(* Logix 5000 project; controller SX_V040001_C001 vendor 1 type 14 code 77 rev 16.23; software revision 16.04; part 11 of 35 *)
(* tags used below, declared in another part *)
   ALL_KINDS : INT[90];
   Basic : INT;
   DRIVE : INT[32];
   DRIVE_INTERVAL : INT[8];
   EMPTYING : INT[18];
   G_AOutput : DINT[8];
   G_DInput : DINT[3];
   G_DOutput : DINT[3];
   METERING : INT[44];
   METERING_PULSE : DINT[14];
   negi_param398 : DINT;
   NOTDOS : INT[6];
   PARAMETER : INT[501];
   T_ACT_DATA_RESET : TIMER;
   T_CHOCO_PRESS_LOW : TIMER;
   T_DEL_DATA : TIMER;
   T_OUTLET_CLOSE : TIMER;
   T_RUN_OUT_CHOCOPUMP : TIMER;
(* MainProgram, continued *)

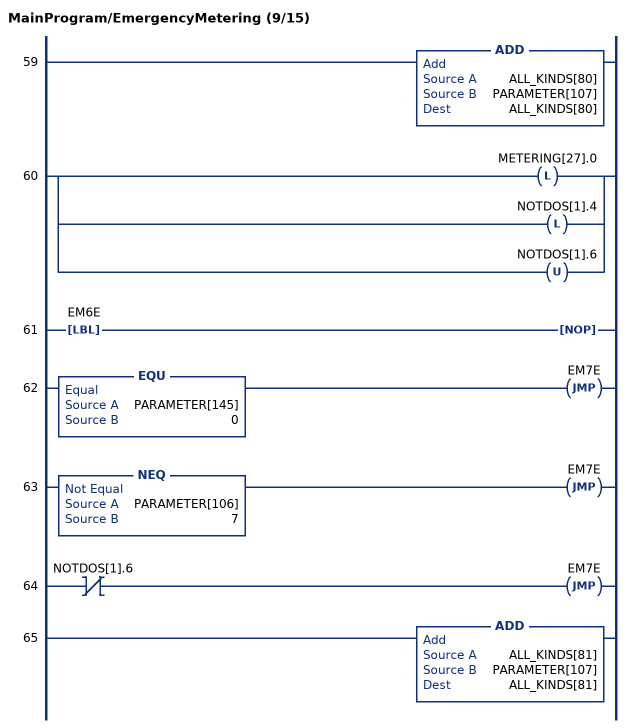
   [picture p232: MainProgram/EmergencyMetering rungs 59-65]
   59: ADD(ALL_KINDS[80],PARAMETER[107],ALL_KINDS[80]);
   60: [OTL(METERING[27].0) ,OTL(NOTDOS[1].4) ,OTU(NOTDOS[1].6) ];
   61: LBL(EM6E)NOP();
   62: EQU(PARAMETER[145],0)JMP(EM7E);
   63: NEQ(PARAMETER[106],7)JMP(EM7E);
   64: XIO(NOTDOS[1].6)JMP(EM7E);
   65: ADD(ALL_KINDS[81],PARAMETER[107],ALL_KINDS[81]);
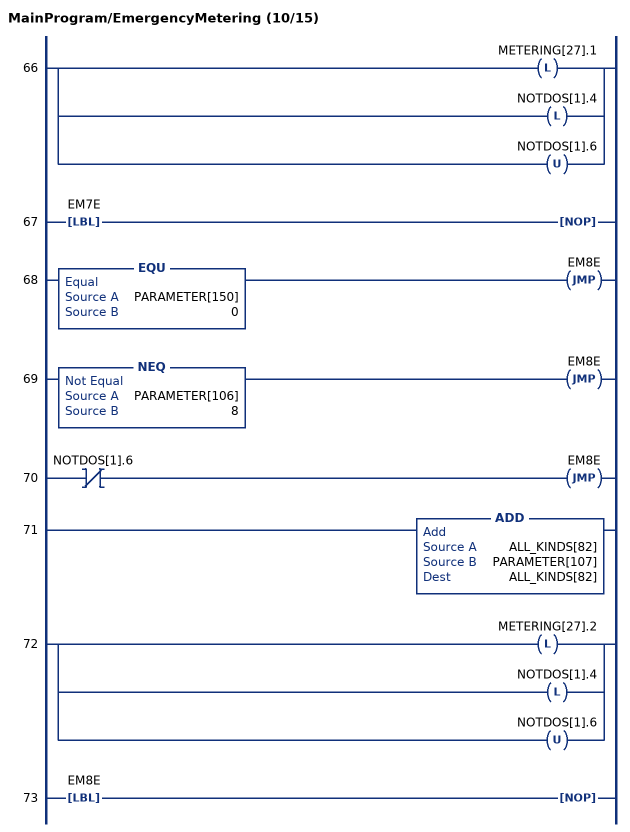
   66: [OTL(METERING[27].1) ,OTL(NOTDOS[1].4) ,OTU(NOTDOS[1].6) ];
   67: LBL(EM7E)NOP();
   68: EQU(PARAMETER[150],0)JMP(EM8E);
   69: NEQ(PARAMETER[106],8)JMP(EM8E);
   70: XIO(NOTDOS[1].6)JMP(EM8E);
   71: ADD(ALL_KINDS[82],PARAMETER[107],ALL_KINDS[82]);
   72: [OTL(METERING[27].2) ,OTL(NOTDOS[1].4) ,OTU(NOTDOS[1].6) ];
   73: LBL(EM8E)NOP();
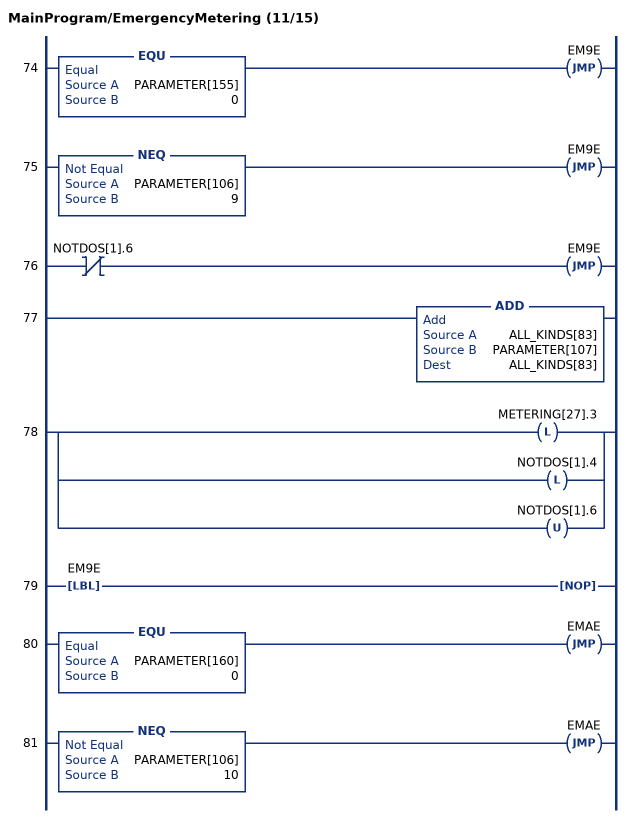
   74: EQU(PARAMETER[155],0)JMP(EM9E);
   75: NEQ(PARAMETER[106],9)JMP(EM9E);
   76: XIO(NOTDOS[1].6)JMP(EM9E);
   77: ADD(ALL_KINDS[83],PARAMETER[107],ALL_KINDS[83]);
   78: [OTL(METERING[27].3) ,OTL(NOTDOS[1].4) ,OTU(NOTDOS[1].6) ];
   79: LBL(EM9E)NOP();
   80: EQU(PARAMETER[160],0)JMP(EMAE);
   81: NEQ(PARAMETER[106],10)JMP(EMAE);
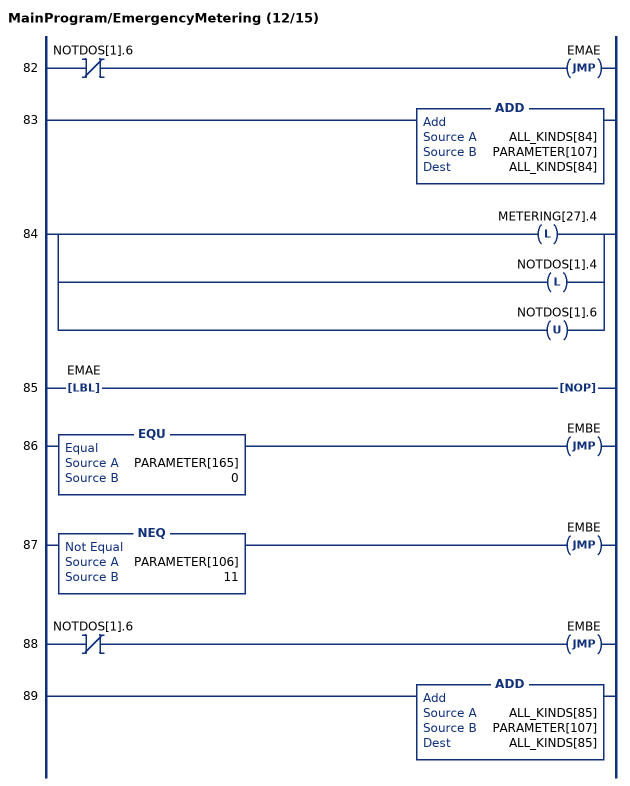
   82: XIO(NOTDOS[1].6)JMP(EMAE);
   83: ADD(ALL_KINDS[84],PARAMETER[107],ALL_KINDS[84]);
   84: [OTL(METERING[27].4) ,OTL(NOTDOS[1].4) ,OTU(NOTDOS[1].6) ];
   85: LBL(EMAE)NOP();
   86: EQU(PARAMETER[165],0)JMP(EMBE);
   87: NEQ(PARAMETER[106],11)JMP(EMBE);
   88: XIO(NOTDOS[1].6)JMP(EMBE);
   89: ADD(ALL_KINDS[85],PARAMETER[107],ALL_KINDS[85]);
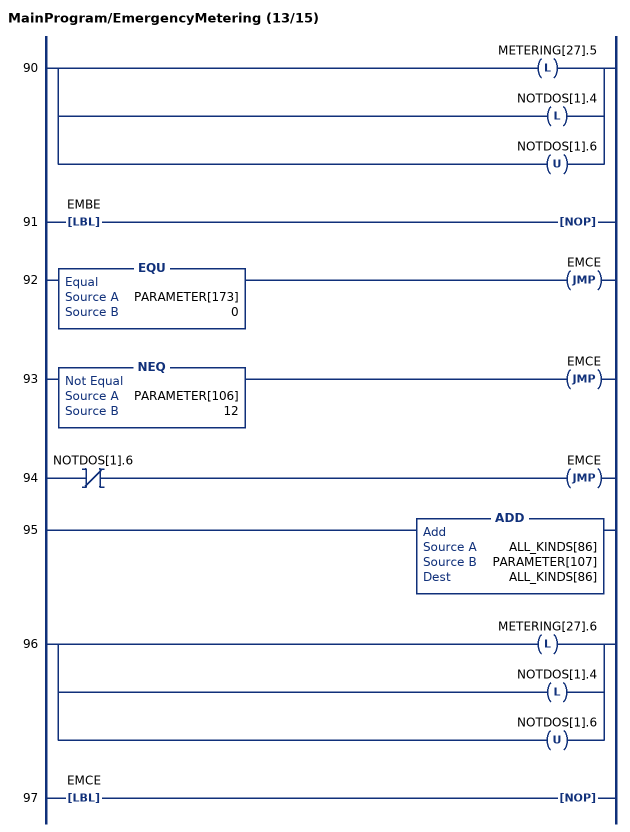
   90: [OTL(METERING[27].5) ,OTL(NOTDOS[1].4) ,OTU(NOTDOS[1].6) ];
   91: LBL(EMBE)NOP();
   92: EQU(PARAMETER[173],0)JMP(EMCE);
   93: NEQ(PARAMETER[106],12)JMP(EMCE);
   94: XIO(NOTDOS[1].6)JMP(EMCE);
   95: ADD(ALL_KINDS[86],PARAMETER[107],ALL_KINDS[86]);
   96: [OTL(METERING[27].6) ,OTL(NOTDOS[1].4) ,OTU(NOTDOS[1].6) ];
   97: LBL(EMCE)NOP();
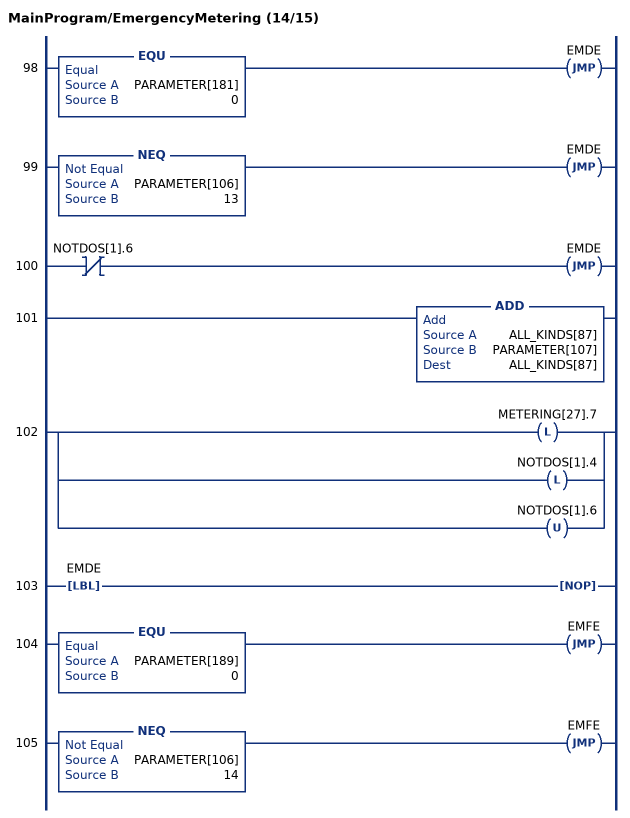
   98: EQU(PARAMETER[181],0)JMP(EMDE);
   99: NEQ(PARAMETER[106],13)JMP(EMDE);
   100: XIO(NOTDOS[1].6)JMP(EMDE);
   101: ADD(ALL_KINDS[87],PARAMETER[107],ALL_KINDS[87]);
   102: [OTL(METERING[27].7) ,OTL(NOTDOS[1].4) ,OTU(NOTDOS[1].6) ];
   103: LBL(EMDE)NOP();
   104: EQU(PARAMETER[189],0)JMP(EMFE);
   105: NEQ(PARAMETER[106],14)JMP(EMFE);
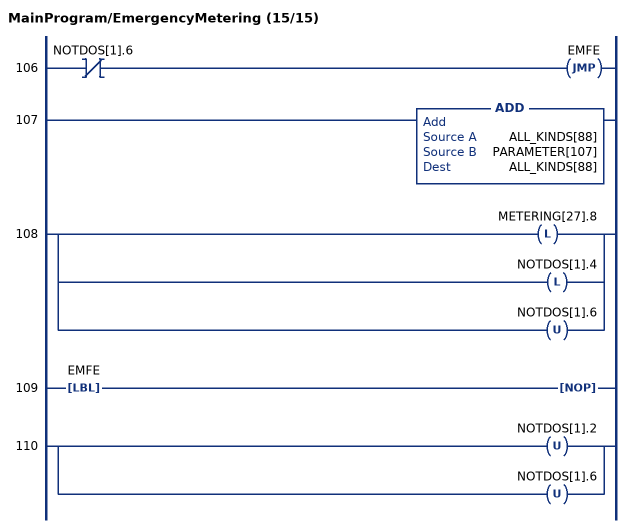
   106: XIO(NOTDOS[1].6)JMP(EMFE);
   107: ADD(ALL_KINDS[88],PARAMETER[107],ALL_KINDS[88]);
   108: [OTL(METERING[27].8) ,OTL(NOTDOS[1].4) ,OTU(NOTDOS[1].6) ];
   109: LBL(EMFE)NOP();
   110: [OTU(NOTDOS[1].2) ,OTU(NOTDOS[1].6) ];
END_ROUTINE

ROUTINE Emptying   (* ladder *)
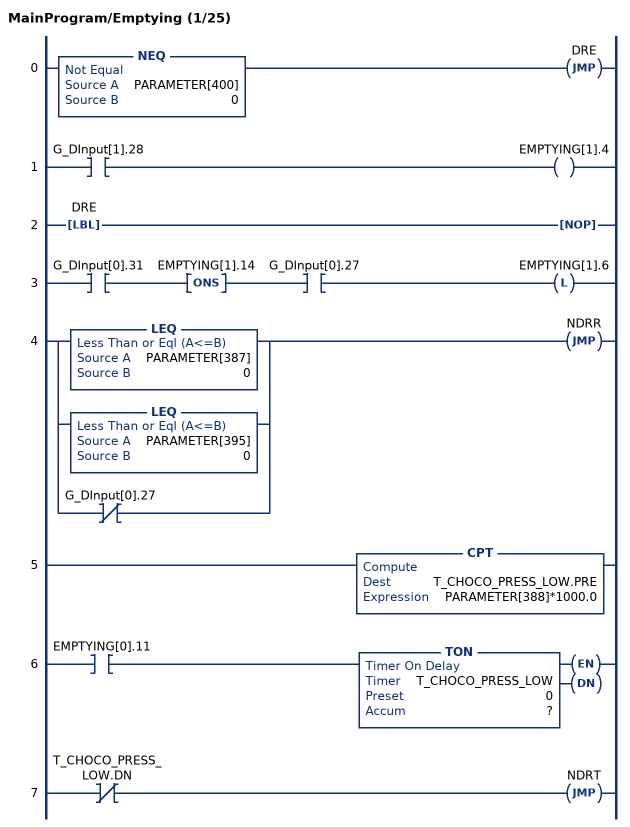
   0: NEQ(PARAMETER[400],0)JMP(DRE);
   1: XIC(G_DInput[1].28)OTE(EMPTYING[1].4);
   2: LBL(DRE)NOP();
   3: XIC(G_DInput[0].31)ONS(EMPTYING[1].14)XIC(G_DInput[0].27)OTL(EMPTYING[1].6);
   4: [LEQ(PARAMETER[387],0) ,LEQ(PARAMETER[395],0) ,XIO(G_DInput[0].27) ]JMP(NDRR);
   5: CPT(T_CHOCO_PRESS_LOW.PRE,PARAMETER[388]*1000.0);
   6: XIC(EMPTYING[0].11)TON(T_CHOCO_PRESS_LOW,?,?);
   7: XIO(T_CHOCO_PRESS_LOW.DN)JMP(NDRT);
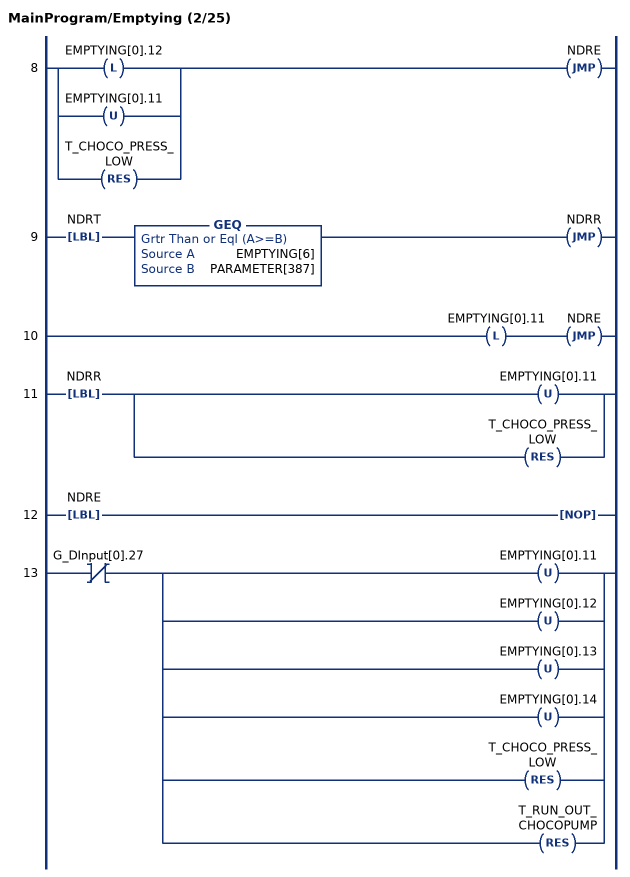
   8: [OTL(EMPTYING[0].12) ,OTU(EMPTYING[0].11) ,RES(T_CHOCO_PRESS_LOW) ]JMP(NDRE);
   9: LBL(NDRT)GEQ(EMPTYING[6],PARAMETER[387])JMP(NDRR);
   10: OTL(EMPTYING[0].11)JMP(NDRE);
   11: LBL(NDRR)[OTU(EMPTYING[0].11) ,RES(T_CHOCO_PRESS_LOW) ];
   12: LBL(NDRE)NOP();
   13: XIO(G_DInput[0].27)[OTU(EMPTYING[0].11) ,OTU(EMPTYING[0].12) ,OTU(EMPTYING[0].13) ,OTU(EMPTYING[0].14) ,RES(T_CHOCO_PRESS_LOW) ,RES(T_RUN_OUT_CHOCOPUMP) ];
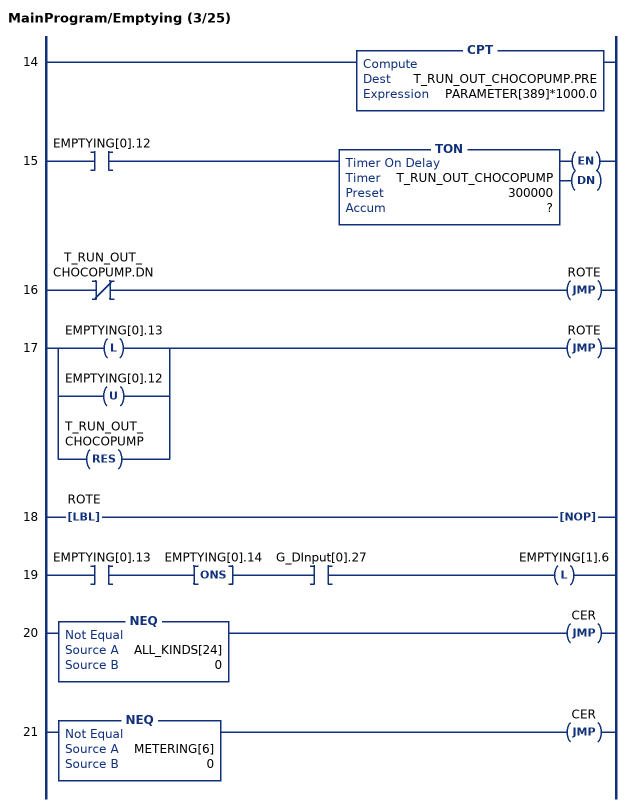
   14: CPT(T_RUN_OUT_CHOCOPUMP.PRE,PARAMETER[389]*1000.0);
   15: XIC(EMPTYING[0].12)TON(T_RUN_OUT_CHOCOPUMP,?,?);
   16: XIO(T_RUN_OUT_CHOCOPUMP.DN)JMP(ROTE);
   17: [OTL(EMPTYING[0].13) ,OTU(EMPTYING[0].12) ,RES(T_RUN_OUT_CHOCOPUMP) ]JMP(ROTE);
   18: LBL(ROTE)NOP();
   19: XIC(EMPTYING[0].13)ONS(EMPTYING[0].14)XIC(G_DInput[0].27)OTL(EMPTYING[1].6);
   20: NEQ(ALL_KINDS[24],0)JMP(CER);
   21: NEQ(METERING[6],0)JMP(CER);
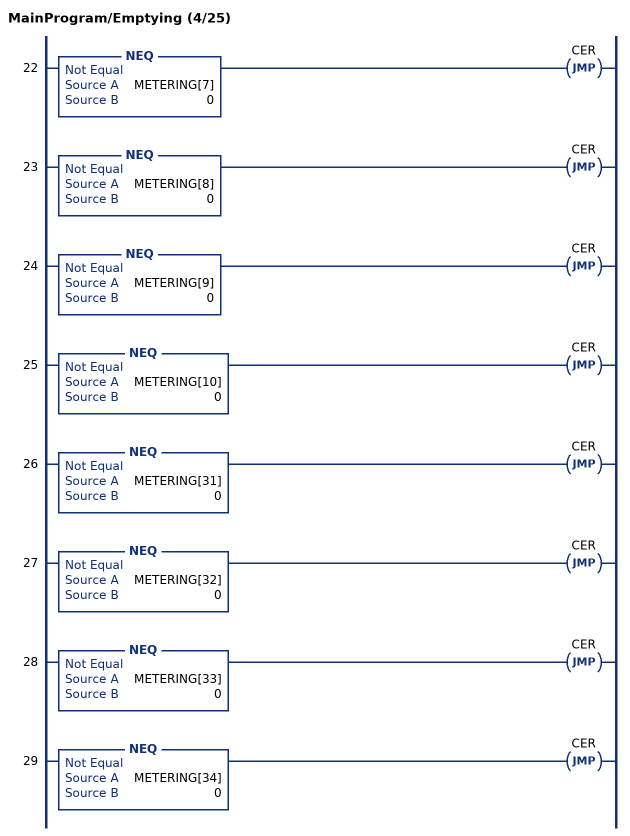
   22: NEQ(METERING[7],0)JMP(CER);
   23: NEQ(METERING[8],0)JMP(CER);
   24: NEQ(METERING[9],0)JMP(CER);
   25: NEQ(METERING[10],0)JMP(CER);
   26: NEQ(METERING[31],0)JMP(CER);
   27: NEQ(METERING[32],0)JMP(CER);
   28: NEQ(METERING[33],0)JMP(CER);
   29: NEQ(METERING[34],0)JMP(CER);
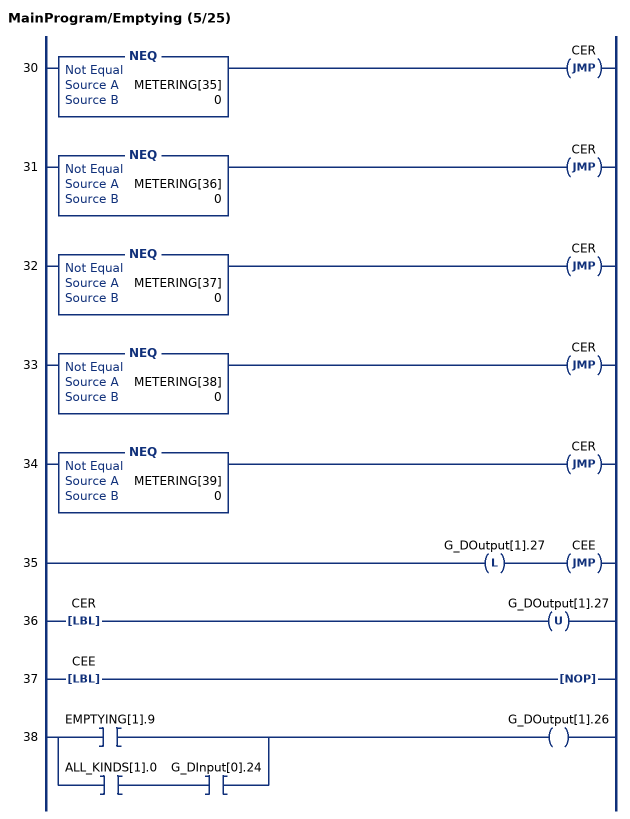
   30: NEQ(METERING[35],0)JMP(CER);
   31: NEQ(METERING[36],0)JMP(CER);
   32: NEQ(METERING[37],0)JMP(CER);
   33: NEQ(METERING[38],0)JMP(CER);
   34: NEQ(METERING[39],0)JMP(CER);
   35: OTL(G_DOutput[1].27)JMP(CEE);
   36: LBL(CER)OTU(G_DOutput[1].27);
   37: LBL(CEE)NOP();
   38: [XIC(EMPTYING[1].9) ,XIC(ALL_KINDS[1].0) XIC(G_DInput[0].24) ]OTE(G_DOutput[1].26);
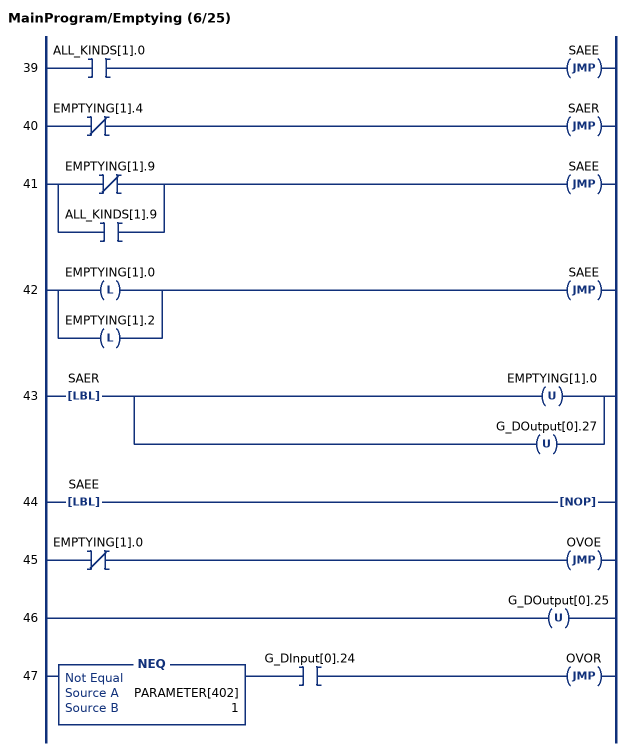
   39: XIC(ALL_KINDS[1].0)JMP(SAEE);
   40: XIO(EMPTYING[1].4)JMP(SAER);
   41: [XIO(EMPTYING[1].9) ,XIC(ALL_KINDS[1].9) ]JMP(SAEE);
   42: [OTL(EMPTYING[1].0) ,OTL(EMPTYING[1].2) ]JMP(SAEE);
   43: LBL(SAER)[OTU(EMPTYING[1].0) ,OTU(G_DOutput[0].27) ];
   44: LBL(SAEE)NOP();
   45: XIO(EMPTYING[1].0)JMP(OVOE);
   46: OTU(G_DOutput[0].25);
   47: NEQ(PARAMETER[402],1)XIC(G_DInput[0].24)JMP(OVOR);
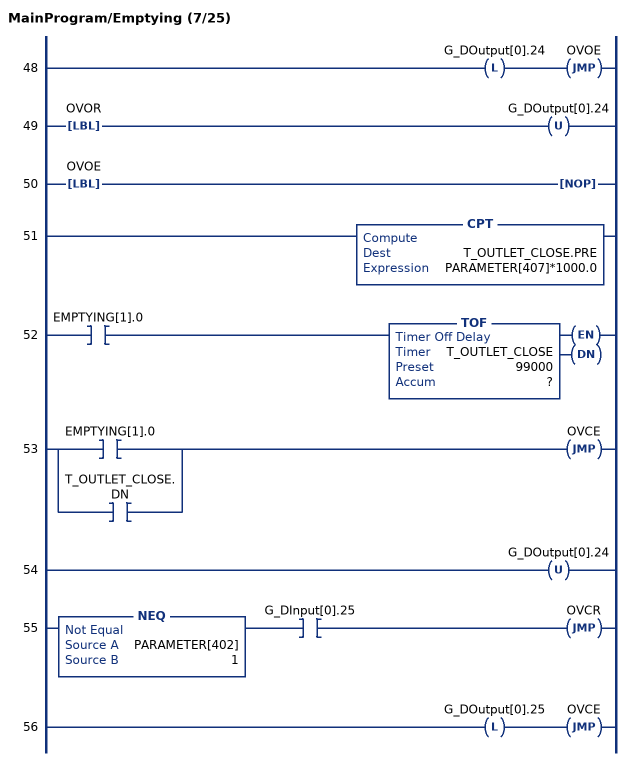
   48: OTL(G_DOutput[0].24)JMP(OVOE);
   49: LBL(OVOR)OTU(G_DOutput[0].24);
   50: LBL(OVOE)NOP();
   51: CPT(T_OUTLET_CLOSE.PRE,PARAMETER[407]*1000.0);
   52: XIC(EMPTYING[1].0)TOF(T_OUTLET_CLOSE,?,?);
   53: [XIC(EMPTYING[1].0) ,XIC(T_OUTLET_CLOSE.DN) ]JMP(OVCE);
   54: OTU(G_DOutput[0].24);
   55: NEQ(PARAMETER[402],1)XIC(G_DInput[0].25)JMP(OVCR);
   56: OTL(G_DOutput[0].25)JMP(OVCE);
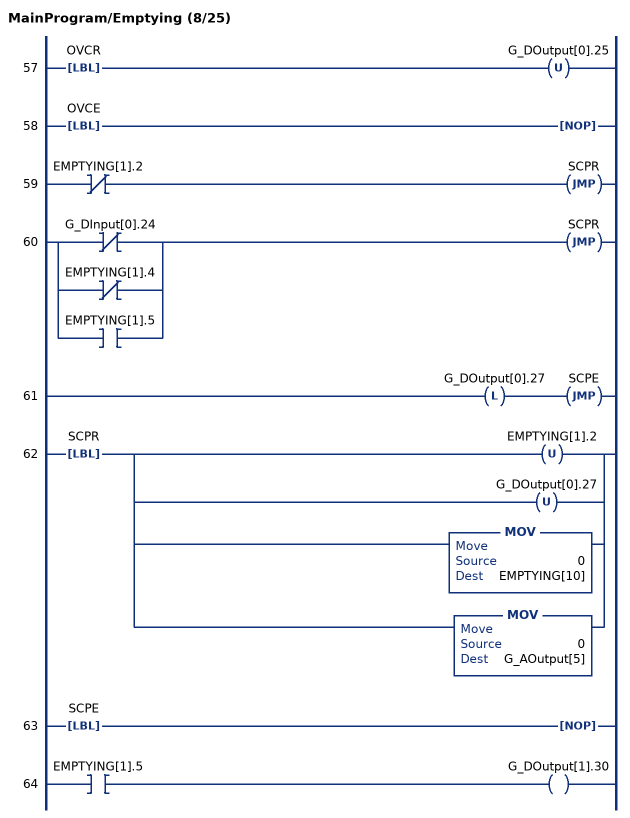
   57: LBL(OVCR)OTU(G_DOutput[0].25);
   58: LBL(OVCE)NOP();
   59: XIO(EMPTYING[1].2)JMP(SCPR);
   60: [XIO(G_DInput[0].24) ,XIO(EMPTYING[1].4) ,XIC(EMPTYING[1].5) ]JMP(SCPR);
   61: OTL(G_DOutput[0].27)JMP(SCPE);
   62: LBL(SCPR)[OTU(EMPTYING[1].2) ,OTU(G_DOutput[0].27) ,MOV(0,EMPTYING[10]) ,MOV(0,G_AOutput[5]) ];
   63: LBL(SCPE)NOP();
   64: XIC(EMPTYING[1].5)OTE(G_DOutput[1].30);
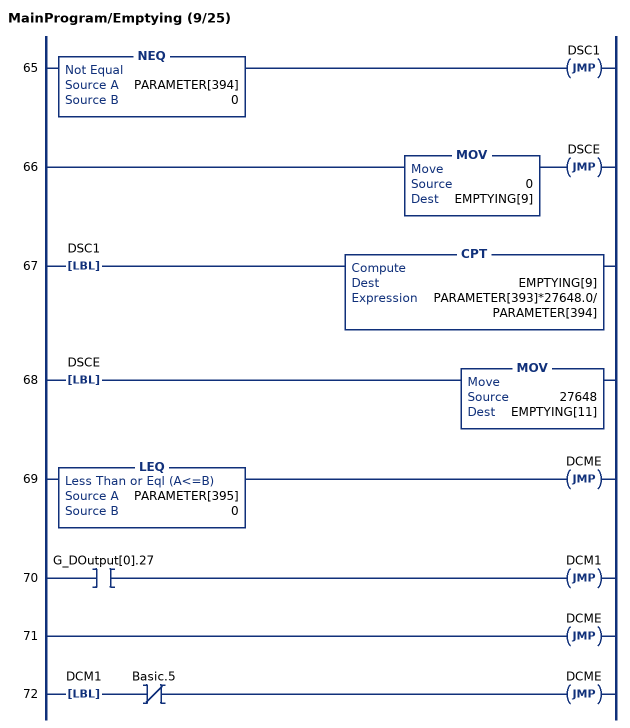
   65: NEQ(PARAMETER[394],0)JMP(DSC1);
   66: MOV(0,EMPTYING[9])JMP(DSCE);
   67: LBL(DSC1)CPT(EMPTYING[9],PARAMETER[393]*27648.0/PARAMETER[394]);
   68: LBL(DSCE)MOV(27648,EMPTYING[11]);
   69: LEQ(PARAMETER[395],0)JMP(DCME);
   70: XIC(G_DOutput[0].27)JMP(DCM1);
   71: JMP(DCME);
   72: LBL(DCM1)XIO(Basic.5)JMP(DCME);
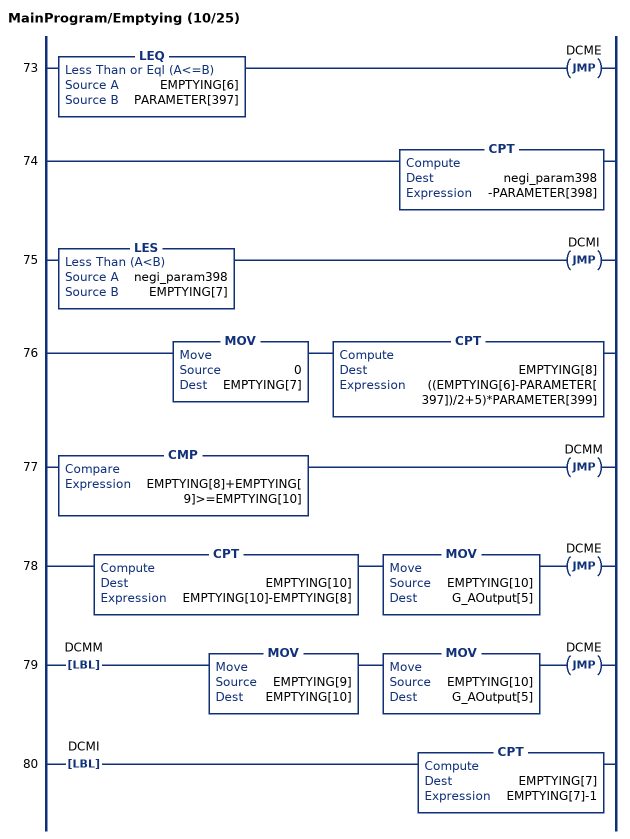
   73: LEQ(EMPTYING[6],PARAMETER[397])JMP(DCME);
   74: CPT(negi_param398,-PARAMETER[398]);
   75: LES(negi_param398,EMPTYING[7])JMP(DCMI);
   76: MOV(0,EMPTYING[7])CPT(EMPTYING[8],((EMPTYING[6]-PARAMETER[397])/2+5)*PARAMETER[399]);
   77: CMP(EMPTYING[8]+EMPTYING[9]>=EMPTYING[10])JMP(DCMM);
   78: CPT(EMPTYING[10],EMPTYING[10]-EMPTYING[8])MOV(EMPTYING[10],G_AOutput[5])JMP(DCME);
   79: LBL(DCMM)MOV(EMPTYING[9],EMPTYING[10])MOV(EMPTYING[10],G_AOutput[5])JMP(DCME);
   80: LBL(DCMI)CPT(EMPTYING[7],EMPTYING[7]-1);
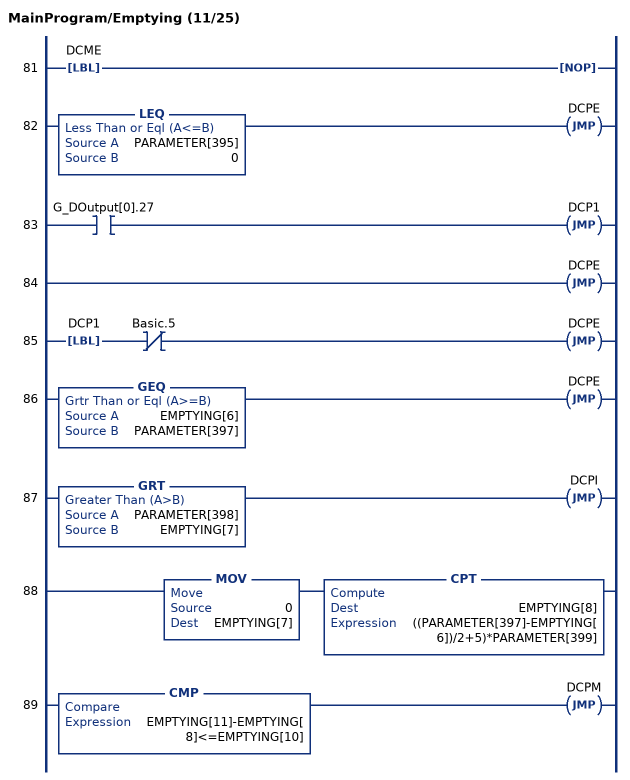
   81: LBL(DCME)NOP();
   82: LEQ(PARAMETER[395],0)JMP(DCPE);
   83: XIC(G_DOutput[0].27)JMP(DCP1);
   84: JMP(DCPE);
   85: LBL(DCP1)XIO(Basic.5)JMP(DCPE);
   86: GEQ(EMPTYING[6],PARAMETER[397])JMP(DCPE);
   87: GRT(PARAMETER[398],EMPTYING[7])JMP(DCPI);
   88: MOV(0,EMPTYING[7])CPT(EMPTYING[8],((PARAMETER[397]-EMPTYING[6])/2+5)*PARAMETER[399]);
   89: CMP(EMPTYING[11]-EMPTYING[8]<=EMPTYING[10])JMP(DCPM);
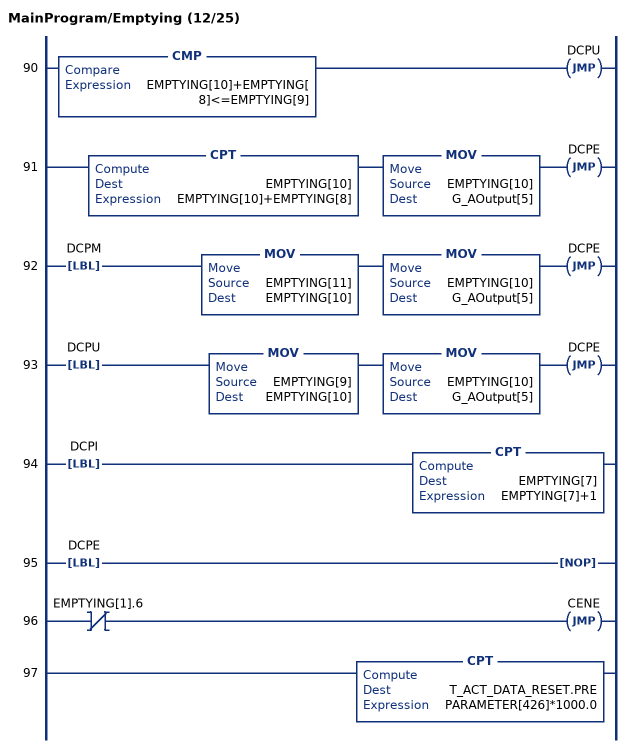
   90: CMP(EMPTYING[10]+EMPTYING[8]<=EMPTYING[9])JMP(DCPU);
   91: CPT(EMPTYING[10],EMPTYING[10]+EMPTYING[8])MOV(EMPTYING[10],G_AOutput[5])JMP(DCPE);
   92: LBL(DCPM)MOV(EMPTYING[11],EMPTYING[10])MOV(EMPTYING[10],G_AOutput[5])JMP(DCPE);
   93: LBL(DCPU)MOV(EMPTYING[9],EMPTYING[10])MOV(EMPTYING[10],G_AOutput[5])JMP(DCPE);
   94: LBL(DCPI)CPT(EMPTYING[7],EMPTYING[7]+1);
   95: LBL(DCPE)NOP();
   96: XIO(EMPTYING[1].6)JMP(CENE);
   97: CPT(T_ACT_DATA_RESET.PRE,PARAMETER[426]*1000.0);
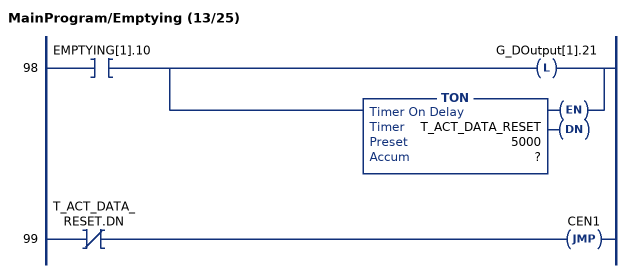
   98: XIC(EMPTYING[1].10)[OTL(G_DOutput[1].21) ,TON(T_ACT_DATA_RESET,?,?) ];
   99: XIO(T_ACT_DATA_RESET.DN)JMP(CEN1);
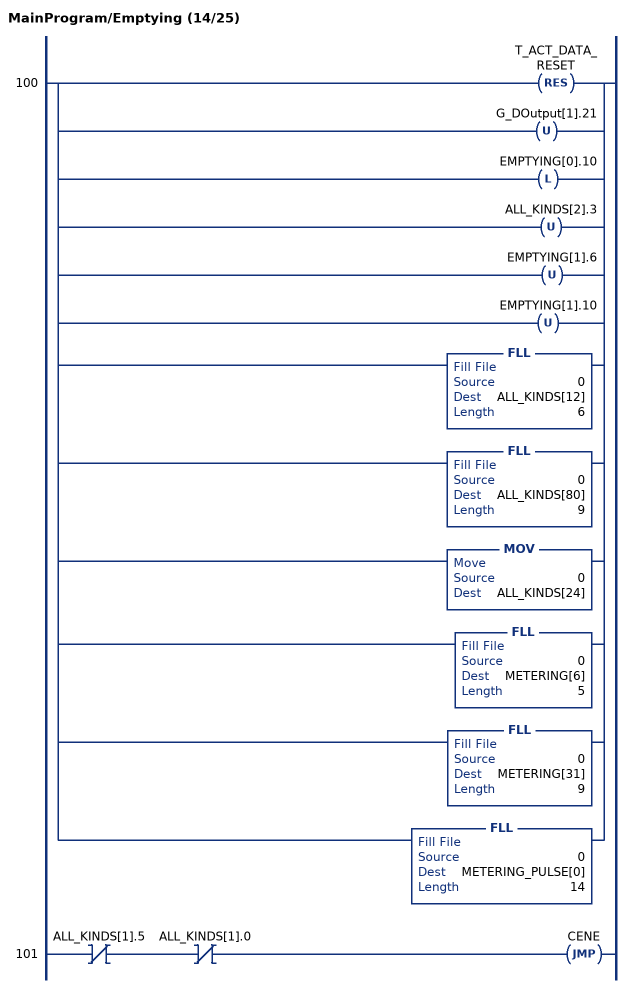
   100: [RES(T_ACT_DATA_RESET) ,OTU(G_DOutput[1].21) ,OTL(EMPTYING[0].10) ,OTU(ALL_KINDS[2].3) ,OTU(EMPTYING[1].6) ,OTU(EMPTYING[1].10) ,FLL(0,ALL_KINDS[12],6) ,FLL(0,ALL_KINDS[80],9) ,MOV(0,ALL_KINDS[24]) ,FLL(0,METERING[6],5) ,FLL(0,METERING[31],9) ,FLL(0,METERING_PULSE[0],14) ];
   101: XIO(ALL_KINDS[1].5)XIO(ALL_KINDS[1].0)JMP(CENE);
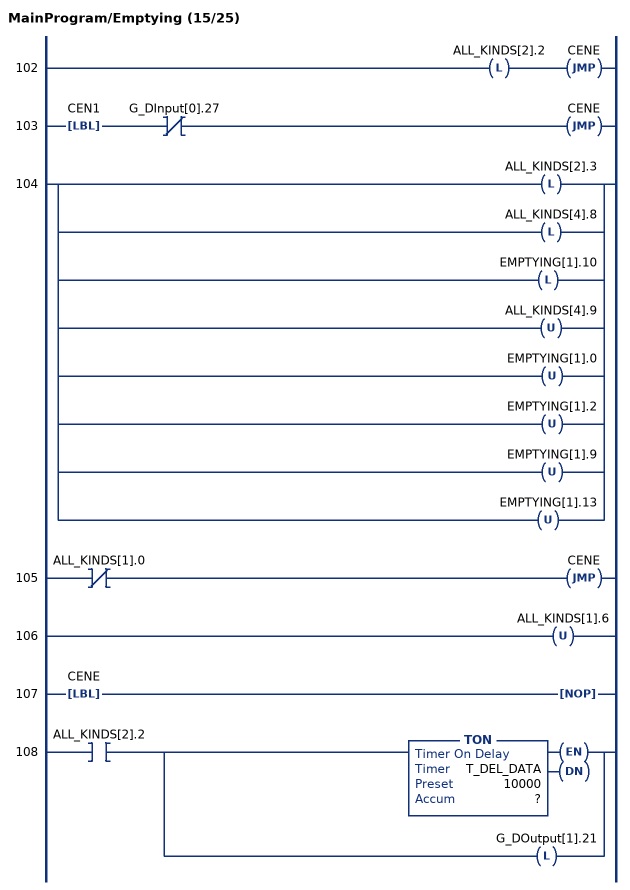
   102: OTL(ALL_KINDS[2].2)JMP(CENE);
   103: LBL(CEN1)XIO(G_DInput[0].27)JMP(CENE);
   104: [OTL(ALL_KINDS[2].3) ,OTL(ALL_KINDS[4].8) ,OTL(EMPTYING[1].10) ,OTU(ALL_KINDS[4].9) ,OTU(EMPTYING[1].0) ,OTU(EMPTYING[1].2) ,OTU(EMPTYING[1].9) ,OTU(EMPTYING[1].13) ];
   105: XIO(ALL_KINDS[1].0)JMP(CENE);
   106: OTU(ALL_KINDS[1].6);
   107: LBL(CENE)NOP();
   108: XIC(ALL_KINDS[2].2)[TON(T_DEL_DATA,?,?) ,OTL(G_DOutput[1].21) ];
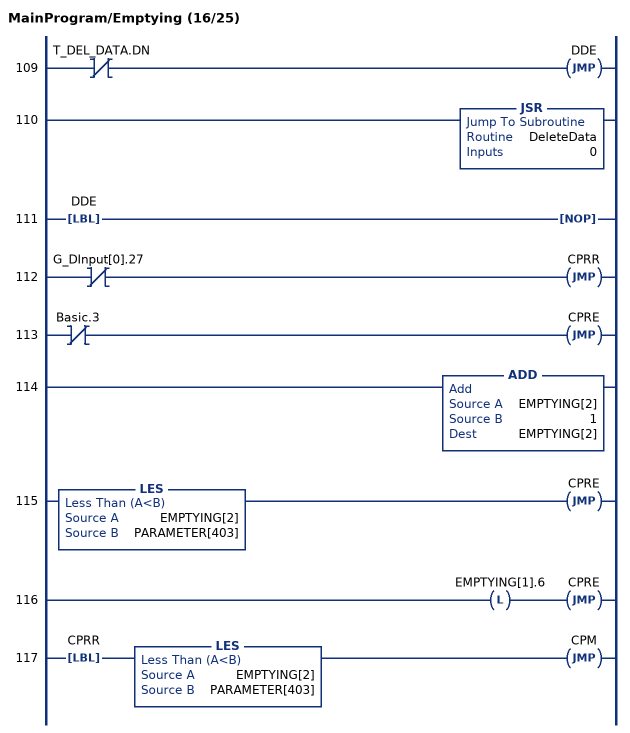
   109: XIO(T_DEL_DATA.DN)JMP(DDE);
   110: JSR(DeleteData,0);
   111: LBL(DDE)NOP();
   112: XIO(G_DInput[0].27)JMP(CPRR);
   113: XIO(Basic.3)JMP(CPRE);
   114: ADD(EMPTYING[2],1,EMPTYING[2]);
   115: LES(EMPTYING[2],PARAMETER[403])JMP(CPRE);
   116: OTL(EMPTYING[1].6)JMP(CPRE);
   117: LBL(CPRR)LES(EMPTYING[2],PARAMETER[403])JMP(CPM);
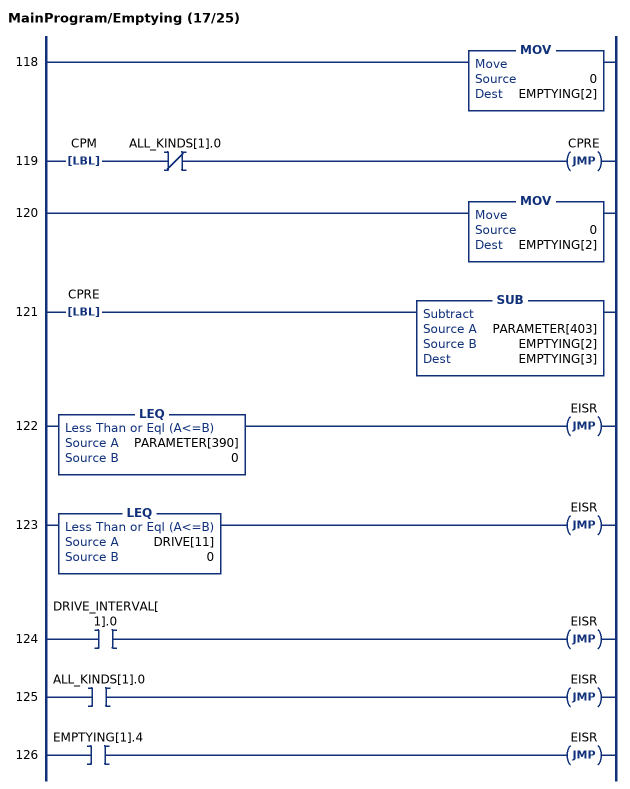
   118: MOV(0,EMPTYING[2]);
   119: LBL(CPM)XIO(ALL_KINDS[1].0)JMP(CPRE);
   120: MOV(0,EMPTYING[2]);
   121: LBL(CPRE)SUB(PARAMETER[403],EMPTYING[2],EMPTYING[3]);
   122: LEQ(PARAMETER[390],0)JMP(EISR);
   123: LEQ(DRIVE[11],0)JMP(EISR);
   124: XIC(DRIVE_INTERVAL[1].0)JMP(EISR);
   125: XIC(ALL_KINDS[1].0)JMP(EISR);
   126: XIC(EMPTYING[1].4)JMP(EISR);
